# EPICS IOC start-up script: iocs/NPDriveExample/iocBoot/iocNPDriveExample/settings.iocsh
# Shell prompt
epicsEnvSet("IOCSH_PS1", "$(IOC)>")

# Prefix used for all PVs in this IOC
epicsEnvSet("PREFIX", "NPDriveExample:")

# Search path for lua scripts
epicsEnvSet("LUA_SCRIPT_PATH", "./scripts")

# Specify largest array CA will transport
# Note for N doubles, need N*8 bytes+some overhead
epicsEnvSet("EPICS_CA_MAX_ARRAY_BYTES", 64010)
